// TIA Portal V15.1 export
// export: Created 2020-06-12T07:35:56.0224609Z, ExportSetting None, DisplayName Totally Integrated Automation Portal, DisplayVersion V15.1, DisplayName TIA Portal Openness, DisplayVersion V15.1, DisplayName STEP 7 Professional, DisplayVersion V15.1, DisplayName STEP 7 Safety, DisplayVersion V15.1, DisplayName WinCC Advanced, DisplayVersion V15.1
FUNCTION "Fake_Input" : Void   // FC133, FBD
{ S7_Optimized_Access := 'TRUE' }
// stored: SetENOAutomatically False
   VAR_TEMP
      tFeederSpeed : Real;
      tMotorSpeed : Real;
   END_VAR
BEGIN

REGION Network 1: ES1LA1.WT01 Simulation [1]
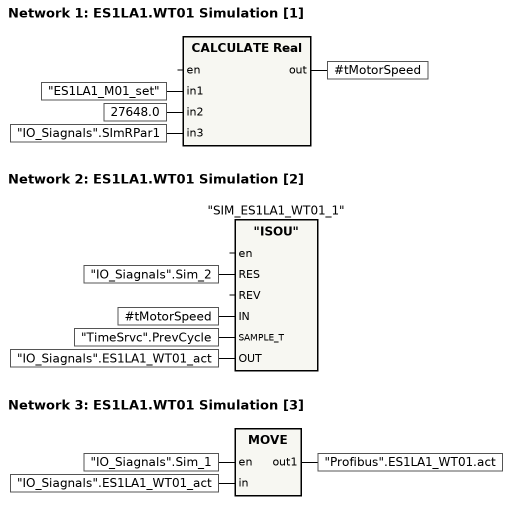
   #tMotorSpeed := "ES1LA1_M01_set"*"IO_Siagnals".SImRPar1/27648.0;
END_REGION

REGION Network 2: ES1LA1.WT01 Simulation [2]
   "SIM_ES1LA1_WT01_1"(RES := "IO_Siagnals".Sim_2,   // "ISOU"
                       IN := #tMotorSpeed,
                       SAMPLE_T := "TimeSrvc".PrevCycle,
                       OUT := "IO_Siagnals".ES1LA1_WT01_act);
END_REGION

REGION Network 3: ES1LA1.WT01 Simulation [3]
   IF "IO_Siagnals".Sim_1 THEN "Profibus".ES1LA1_WT01.act := "IO_Siagnals".ES1LA1_WT01_act; END_IF;
END_REGION
END_FUNCTION
